(* IEC 61131-3 sources: plc-vscode/tests/st/test-ready/trust-platform/examples/vendor_library_stubs/vendor/siemens, 2 files *)

(* ---- norm_scale.st ---- *)
FUNCTION_BLOCK NORM_X
VAR_INPUT
    X : REAL;
    X_MIN : REAL;
    X_MAX : REAL;
END_VAR
VAR_OUTPUT
    Y : REAL;
END_VAR
END_FUNCTION_BLOCK

FUNCTION_BLOCK SCALE_X
VAR_INPUT
    X : REAL;
    X_MIN : REAL;
    X_MAX : REAL;
    Y_MIN : REAL;
    Y_MAX : REAL;
END_VAR
VAR_OUTPUT
    Y : REAL;
END_VAR
END_FUNCTION_BLOCK

(* ---- tcon.st ---- *)
FUNCTION_BLOCK TCON
VAR_INPUT
    REQ : BOOL;
END_VAR
VAR_OUTPUT
    DONE : BOOL;
    ERROR : BOOL;
    STATUS : WORD;
END_VAR
END_FUNCTION_BLOCK
